(* Logix 5000 project; controller PBS_Perfusion vendor 1 type 14 code 217 rev 32.14; software revision 32.03; part 23 of 27 *)
(* tags used below, declared in another part *)
   Ref_FaultCodeList : P_DescList[1];   // Tag containing List of Fault Codes (DINT) and their Descriptions (STRING)
   Inp_LastFaultCode : DINT;   // Most recent drive fault code (enumeration)
   Inp_Ready : BOOL;   // 1=Drive is ready to run
   Inp_CommandDir : BOOL;   // 1=Drive is commanded Forward, 0=Drive is commanded Reverse
   Inp_IOFault : BOOL;   // Input Communication Status 0=OK, 1=fail
   Inp_Sim : BOOL;   // 1=Simulate working drive; 0=Start/Stop/ Monitor actual drive
   Cfg_HasReverse : BOOL;   // 1=Drive can be run reverse, 0=Forward only
   Cfg_HasJog : BOOL;   // 1=Drive Jog Command enabled/visible, 0=Drive Jog Command not allowed
   Cfg_HasRunFdbk : BOOL;   // 1=Drive provides feedback signal on Inp_Running when running
   Cfg_HasSpeedFdbk : BOOL;   // 1=Drive provides speed feedback on Inp_SpeedFdbk
   Cfg_UseSpeedFdbk : BOOL;   // 1=Drive speed determines running state, 0=state determined by drive Active input bit
   Cfg_HasOutDatalink : BOOL;   // 1=A signal is connected to Out_Datalink
   Cfg_SetTrack : BOOL;   // 1=Settings track for unselected sources, 0=no tracking
   Cfg_SetTrackOvrdHand : BOOL;   // 1=Prog/Oper/Ext Settings track Override/Hand
   Cfg_OperStopPrio : BOOL;   // 1=OCmd_Stop any time, 0=OCmd_Stop only when Oper selected
   Cfg_OCmdResets : BOOL;   // 1=New drive OCmd resets shed latches and cleared alarms, 0=OCmdReset req'd.
   Cfg_ShedOnFailToStart : BOOL;   // 1=Stop Motor and Alarm on Fail to Start; 0=Alarm only on Fail to Start
   Cfg_MinSpdRef : REAL;   // Minimum Speed Reference in EU (for limiting)
   Cfg_MaxSpdRef : REAL;   // Maximum Speed Reference in EU (for limiting)
   Cfg_SpeedRefRawMin : REAL;   // Speed Reference Minimum in Drive (raw) Units (for scaling)
   Cfg_SpeedRefRawMax : REAL;   // Speed Reference Maximum in Drive (raw) Units (for scaling)
   Cfg_SpeedRefEUMin : REAL;   // Speed Reference Minimum in Engineering Units (for scaling)
   Cfg_SpeedRefEUMax : REAL;   // Speed Reference Maximum in Engineering Units (for scaling)
   Cfg_OutDatalinkRawMin : REAL;   // Output Datalink Minimum in Drive (raw) Units (for scaling)
   Cfg_OutDatalinkRawMax : REAL;   // Output Datalink Maximum in Drive (raw) Units (for scaling)
   Cfg_OutDatalinkEUMin : REAL;   // Output Datalink Minimum in Engineering Units (for scaling)
   Cfg_OutDatalinkEUMax : REAL;   // Output Datalink Maximum in Engineering Units (for scaling)
   Cfg_OperKeep : SINT;   // Oper keeps control in Prog / Ext: .0=Reference, .1=Start/Stop/Fwd/ Rev, .3=OutDatalink
   Cfg_ProgKeep : SINT;   // Prog keeps control in Oper / Ext: .0=Reference, .1=Start/Stop/Fwd/ Rev, .3=OutDatalink
   PSet_SpeedRef : REAL;   // Program Setting of Speed Reference (EU)
   PSet_OutDatalink : REAL;   // Program Setting of Output Datalink (EU)
   XSet_SpeedRef : REAL;   // External Setting of Speed Reference (EU)
   XSet_OutDatalink : REAL;   // External Setting of Output Datalink (EU)
   Out_SpeedRef : REAL;   // Drive Speed Reference in Drive Units (typ. 0-32767 = 0 to max freq.)
   Out_Datalink : REAL;   // Auxiliary Signal (datalink) Output in Drive (raw) Units
   Out_Run : BOOL;   // 1=Start/Run Drive, 0=Stop Drive (for held starter type)
   Out_Stop : BOOL;   // 1=Stop Drive, 0=drive left in current state
   Out_Start : BOOL;   // 1=Start Drive, 0=drive left in current state
   Out_Jog : BOOL;   // 1=Jog drive at Jog Speed, -->0=stop jogging
   Out_Fwd : BOOL;   // 1=Set drive direction to Forward
   Out_Rev : BOOL;   // 1=Set drive direction to Reverse
   Out_Horn : BOOL;   // 1=Sound audible prior to commanded motor start
   Val_SpeedRef : REAL;   // Speed Reference (target) to drive
   Val_OutDatalink : REAL;   // Output Datalink value to drive
   Val_LastFaultCode : DINT;   // Most recent drive fault code (enumeration)
   SrcQ_IO : DINT;   // Source and Quality of primary I/O (enumeration)
   SrcQ : DINT;   // Source and Quality of primary Val/Sts (enumeration)
   Val_Cmd : DINT;   // Device Command 0=None, 1=Stop, 2=StartFwd 3=StartRev 4=JogFwd 5=JogRev
   Val_Sts : DINT;   // Device Sts: 0=? 1=Stopped 2=RunFwd 3=RunRev 4=RunSlow 5=StartFwd 6=StartRev 7=StartSlow 8=JogFwd 9=JogRev 10=Stopping
   Val_Fault : DINT;   // Device Fault Status 0=None, 16=Fail to Start, 17 = Fail to Stop, 18=Drive Fault, 32=I/O Fault, 34=Config Error
   Val_NotifyAll : DINT;   // Highest Alarm prio and ack status this object + channel (enum)
   Val_UnackAlmC : DINT;   // Count of Unacknowledged Alarms
   Sts_Stopped : BOOL;   // 1=Drive requested to stop and is confirmed stopped
   Sts_StartingFwd : BOOL;   // 1=Drive requested to run forward and awaiting run feedback
   Sts_StartingRev : BOOL;   // 1=Drive requested to run reverse and awaiting run feedback
   Sts_RunningFwd : BOOL;   // 1=Drive requested to run and is confirmed running forward
   Sts_RunningRev : BOOL;   // 1=Drive requested to run and is confirmed running reverse
   Sts_StoppingFwd : BOOL;   // 1=Drive running forward requested to stop and awaiting stopped feedback
   Sts_StoppingRev : BOOL;   // 1=Drive running reverse requested to stop and awaiting stopped feedback
   Sts_JoggingFwd : BOOL;   // 1=Drive requested to Jog Forward
   Sts_JoggingRev : BOOL;   // 1=Drive requested to Jog Reverse
   Sts_Horn : BOOL;   // 1=Motor Horn Active
   Sts_CommandDir : BOOL;   // 1=Drive commanded to Forward, 0=Reverse
   Sts_ActualDir : BOOL;   // 1=Drive Actual direction is Forward, 0=Reverse
   Sts_SpeedLimited : BOOL;   // 1=Speed Reference Setting exceeds configured Max/Min limit
   Sts_NotRdy : BOOL;   // 1=Device Not Ready, see detail bits for reason
   Nrdy_CfgErr : BOOL;   // 1=Device Not Ready: Configuration Error
   Nrdy_Fail : BOOL;   // 1=Device Not Ready: Device Failure (Shed Requires Reset)
   Nrdy_IOFault : BOOL;   // 1=Device Not Ready: I/O Fault (Shed Requires Reset)
   Nrdy_PrioStop : BOOL;   // 1=Device Not Ready: Oper/Ext Priority Stop Requires Reset
   Nrdy_Trip : BOOL;   // 1=Device not Ready: Deivce Tripped (Drive Fault)
   Sts_AlmInh : BOOL;   // 1=An Alarm is Shelved, Disabled or Suppressed, display icon
   Sts_Err : BOOL;   // 1=Error in Config: see detail bits for reason
   Err_Alarm : BOOL;   // 1=Error in Config: Alarm Min On Time, Shelf Time, Severity
   Err_FdbkRaw : BOOL;   // 1=Erron in Config: Speed Fdbk Raw Min = Max
   Err_FdbkEU : BOOL;   // 1=Error in Config: Speed Fdbk EU Min = Max
   Err_RefEU : BOOL;   // 1=Error in Config: Speed Ref EU Min = Max
   Err_OutDLEU : BOOL;   // 1=Error in Config: Output Datalink EU Min = Max
   Sts_Hand : ALIAS FOR CmdSrc.Sts_Hand;
   Sts_OoS : ALIAS FOR CmdSrc.Sts_OoS;
   Sts_Maint : ALIAS FOR CmdSrc.Sts_Maint;
   Sts_Ovrd : ALIAS FOR CmdSrc.Sts_Ovrd;
   Sts_RdyReset : ALIAS FOR ORdy_Reset;   // 1=A latched alarm or shed condition is ready to be reset
   Sts_RdyAck : BOOL;   // 1=An alarm is ready to be acknowledged
   Sts_FailToStart : ALIAS FOR FailToStart.Inp;   // 1=Drive Failed to Start (One-Shot)
   Sts_FailToStop : ALIAS FOR FailToStop.Inp;   // 1=Drive Failed to Stop
   Sts_DriveFault : ALIAS FOR DriveFault.Inp;   // 1=Drive Fault (see drive display or manual)
   Sts_IOFault : ALIAS FOR IOFault.Inp;   // I/O Comm Fault Status (0=OK, 1=Bad)
   P_VSD : BOOL;   // Unique Parameter Name for auto - discovery
   CmdSrc : P_CmdSrc;   // Drive Mode Selection
   IOFault : P_Alarm;   // I/O Fault Alarm
   IntlkTrip : P_Alarm;   // Interlock Trip Alarm
   FailToStop : P_Alarm;   // Drive Failed to Stop Alarm
   FailToStart : P_Alarm;   // Drive Failed to Start Alarm
   Wrk_Run : BOOL;   // 1=Drive should be "running", 0=should be "stopped"
   Wrk_StartRetrigT : TIMER;   // Time to pulse start output on start command retrigger (Maint)
   Wrk_StopRetrigT : TIMER;   // Time to pulse stop output on stop command retrigger (Maint)
   Wrk_RunFdbk : BOOL;   // Run Feedback based on mode, simulation, etc. 1=running
   Wrk_Notify : DINT;   // Buffer for building Val_Notify
   DriveFault : P_Alarm;   // Drive Faulted Alarm
   Wrk_SpeedRef : REAL;   // Working copy of Speed Reference (for limiting)
   Wrk_Rev : BOOL;   // Working (internal) Direction 1=Reverse 0=Forward (default)
   Wrk_Jog : BOOL;   // 1=Jog Drive, 0=Drive not jogging
   Wrk_OutDatalink : REAL;   // Selected Output Datalink setting
   Wrk_StopT : TIMER;   // Stop Check Timer (for Fail to Stop)
   Wrk_StartT : TIMER;   // Start Check Timer (for Fail to Start)
   Wrk_Cmd : DINT;   // Buffer for building Val_Cmd
   Wrk_Sts : DINT;   // Buffer for building Val_Sts
   Wrk_Fault : DINT;   // Buffer for building Val_Fault
   Wrk_Retrigger : BOOL;   // Maint Start issued while running or Stop while stopped
   Wrk_JogT : TIMER;   // Jog Timer
   Wrk_FaultDescFSC : CONTROL;   // FSC control for Fault Code List search
   Val_FaultDesc : STRING_40;   // Description of Drive Fault (given LastFaultCode)
   Wrk_SrcQ : DINT;   // Register for building Source / Quality enumeration
   Val_Notify : DINT;   // Current Alarm Level and Acknowledgement (enumeration)
   Wrk_NotRdy : BOOL;   // Device Not Ready conditions excluding shed latches
   Wrk_StartInhT : TIMER;   // Local Start Inhibit Timer
   Wrk_StopInhT : TIMER;   // Local Stop Inhibit Timer
   Wrk_Hand : BOOL;   // Perform Hand Mode alignment with actual device state
   Wrk_UnackAlmC : DINT;   // Buffer for building Val_UnackAlmC
   Wrk_StartHornT : TIMER;   // Timer for audible alert or start
   Wrk_StartHorn : BOOL;   // 1=Sound audible prior to commanded motor start
   Wrk_RevPermOK : BOOL;   // Reverse Permissives and NB Permissive OK
   Wrk_FwdPermOK : BOOL;   // Forward Permissives and NB Permissive OK
   OSet_OutDatalink : REAL;   // Operator Setting of Output Datalink (EU)
   OSet_SpeedRef : REAL;   // Operator Setting of Speed Reference (EU)
   ORdy_ResetAckAll : BOOL;   // 1=Ready for OCmd_ResetAckAll (enables HMI button)
   ORdy_Reset : BOOL;   // 1=Ready for OCmd_Reset (enables HMI button)
   ORdy_JogRev : BOOL;   // 1=Ready for OCmd_JogRev (enabled HMI button)
   ORdy_JogFwd : BOOL;   // 1=Ready for OCmd_JogFwd (enables HMI button)
   ORdy_Stop : BOOL;   // 1=Ready for OCmd_Stop (enables HMI button)
   ORdy_StartRev : BOOL;   // 1=Ready for OCmd_StartRev (enables HMI button)
   ORdy_StartFwd : BOOL;   // 1=Ready for OCmd_StartFwd (enables HMI button)
   Wrk_OperHas1 : BOOL;   // Operator has Commands
   REAL : DINT;
(* P_VSD, continued *)

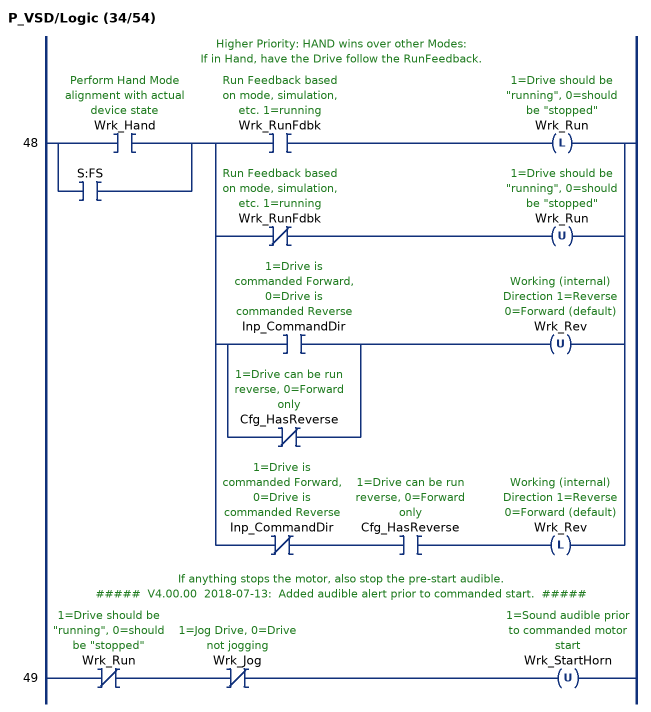
   [picture p515: P_VSD/Logic rungs 48-49]
   // Higher Priority: HAND wins over other Modes:
   // If in Hand, have the Drive follow the RunFeedback.
   48: [XIC(Wrk_Hand) ,XIC(S:FS) ][XIC(Wrk_RunFdbk) OTL(Wrk_Run) ,XIO(Wrk_RunFdbk) OTU(Wrk_Run) ,[XIC(Inp_CommandDir) ,XIO(Cfg_HasReverse) ] OTU(Wrk_Rev) ,XIO(Inp_CommandDir) XIC(Cfg_HasReverse) OTL(Wrk_Rev) ];
   // If anything stops the motor, also stop the pre-start audible.
   // #####  V4.00.00  2018-07-13:  Added audible alert prior to commanded start.  #####
   49: XIO(Wrk_Run)XIO(Wrk_Jog)OTU(Wrk_StartHorn);
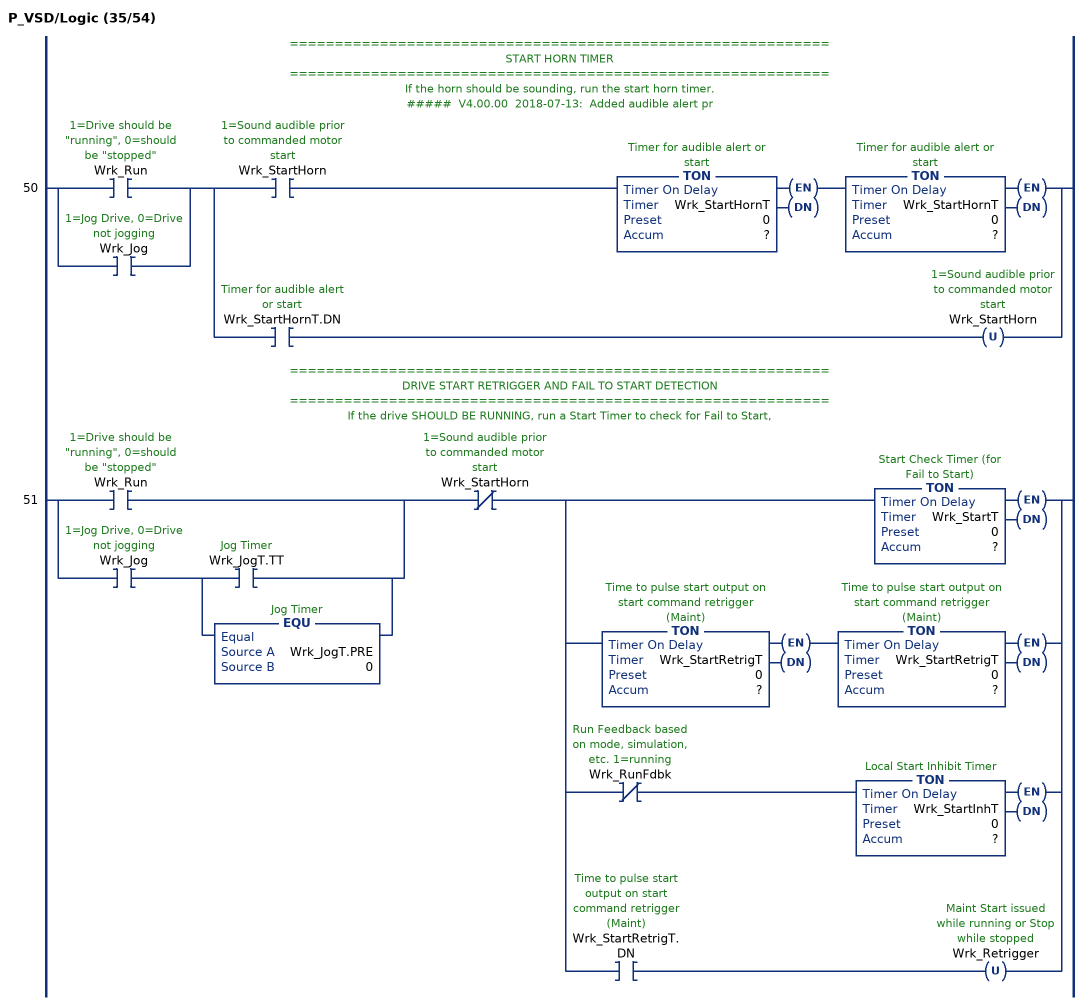
   // ============================================================
   // START HORN TIMER
   // ============================================================
   // If the horn should be sounding, run the start horn timer.
   // #####  V4.00.00  2018-07-13:  Added audible alert pr
   50: [XIC(Wrk_Run) ,XIC(Wrk_Jog) ][XIC(Wrk_StartHorn) TON(Wrk_StartHornT,?,?) TON(Wrk_StartHornT,?,?) ,XIC(Wrk_StartHornT.DN) OTU(Wrk_StartHorn) ];
   // ============================================================
   // DRIVE START RETRIGGER AND FAIL TO START DETECTION
   // ============================================================
   // If the drive SHOULD BE RUNNING, run a Start Timer to check for Fail to Start,
   51: [XIC(Wrk_Run) ,XIC(Wrk_Jog) [XIC(Wrk_JogT.TT) ,EQU(Wrk_JogT.PRE,0) ] ]XIO(Wrk_StartHorn)[TON(Wrk_StartT,?,?) ,TON(Wrk_StartRetrigT,?,?) TON(Wrk_StartRetrigT,?,?) ,XIO(Wrk_RunFdbk) TON(Wrk_StartInhT,?,?) ,XIC(Wrk_StartRetrigT.DN) OTU(Wrk_Retrigger) ];
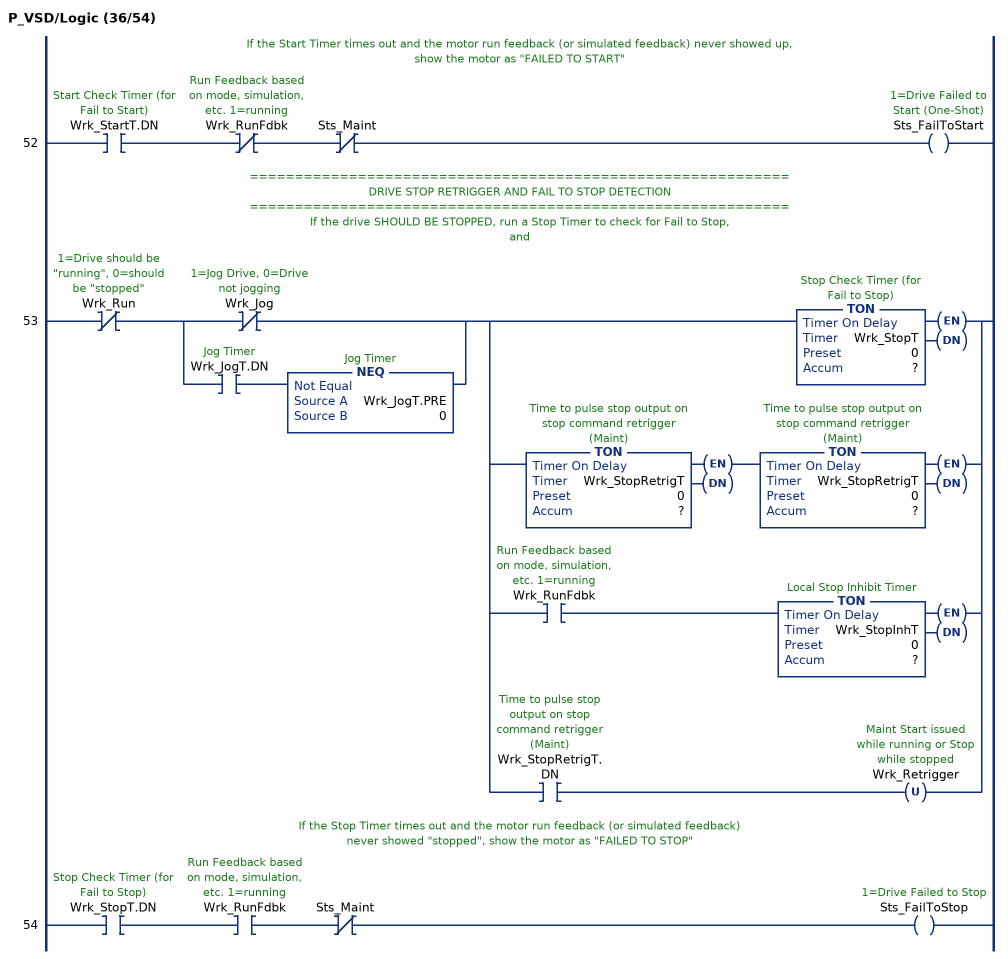
   // If the Start Timer times out and the motor run feedback (or simulated feedback) never showed up,
   // show the motor as "FAILED TO START"
   52: XIC(Wrk_StartT.DN)XIO(Wrk_RunFdbk)XIO(Sts_Maint)OTE(Sts_FailToStart);
   // ============================================================
   // DRIVE STOP RETRIGGER AND FAIL TO STOP DETECTION
   // ============================================================
   // If the drive SHOULD BE STOPPED, run a Stop Timer to check for Fail to Stop,
   //  and
   53: XIO(Wrk_Run)[XIO(Wrk_Jog) ,XIC(Wrk_JogT.DN) NEQ(Wrk_JogT.PRE,0) ][TON(Wrk_StopT,?,?) ,TON(Wrk_StopRetrigT,?,?) TON(Wrk_StopRetrigT,?,?) ,XIC(Wrk_RunFdbk) TON(Wrk_StopInhT,?,?) ,XIC(Wrk_StopRetrigT.DN) OTU(Wrk_Retrigger) ];
   // If the Stop Timer times out and the motor run feedback (or simulated feedback)
   // never showed "stopped", show the motor as "FAILED TO STOP"
   54: XIC(Wrk_StopT.DN)XIC(Wrk_RunFdbk)XIO(Sts_Maint)OTE(Sts_FailToStop);
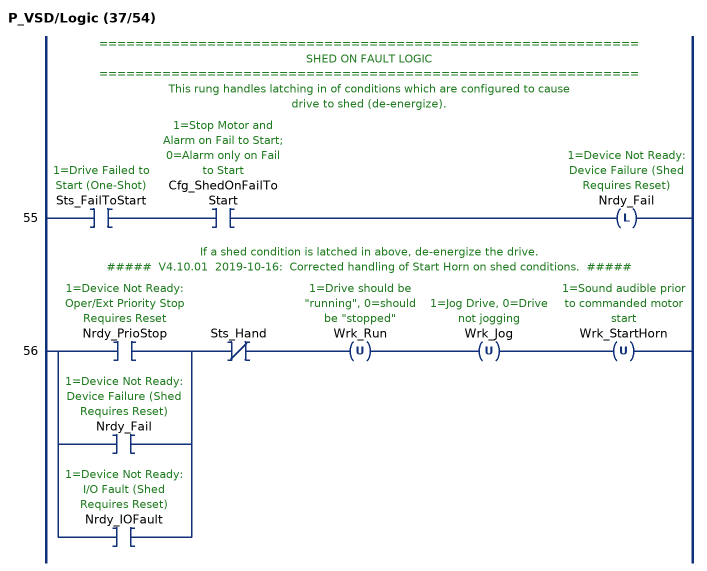
   // ============================================================
   // SHED ON FAULT LOGIC
   // ============================================================
   // This rung handles latching in of conditions which are configured to cause
   // drive to shed (de-energize).
   55: XIC(Sts_FailToStart)XIC(Cfg_ShedOnFailToStart)OTL(Nrdy_Fail);
   // If a shed condition is latched in above, de-energize the drive.
   // #####  V4.10.01  2019-10-16:  Corrected handling of Start Horn on shed conditions.  #####
   56: [XIC(Nrdy_PrioStop) ,XIC(Nrdy_Fail) ,XIC(Nrdy_IOFault) ]XIO(Sts_Hand)OTU(Wrk_Run)OTU(Wrk_Jog)OTU(Wrk_StartHorn);
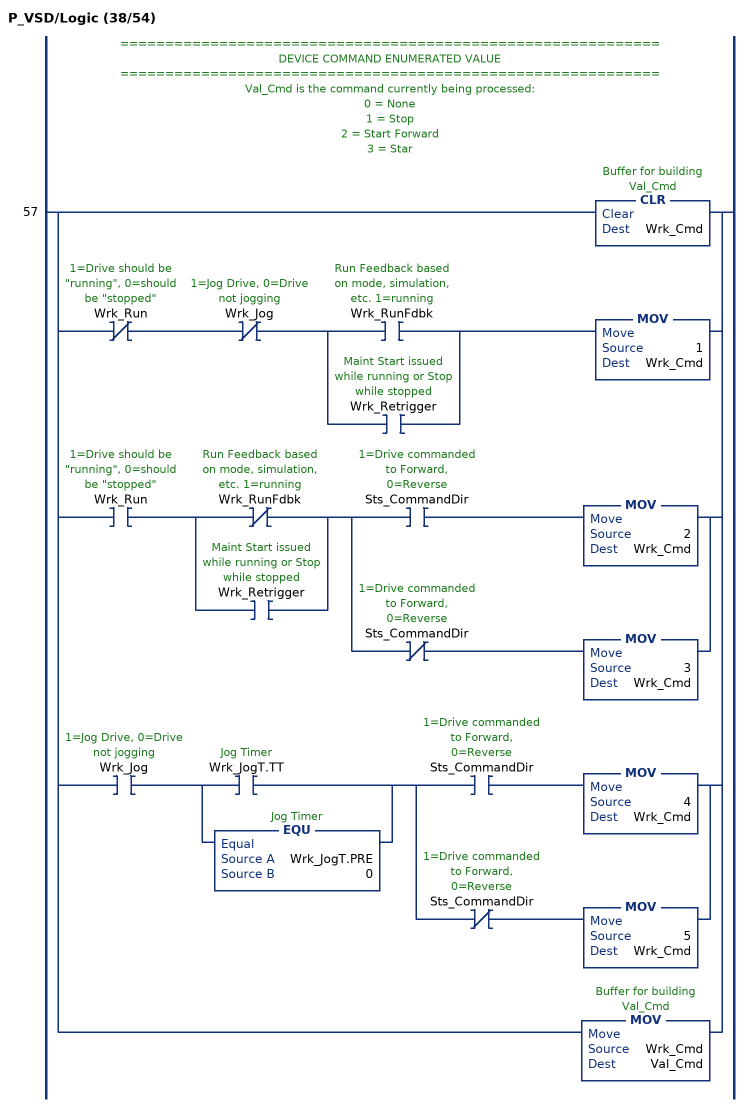
   // ============================================================
   // DEVICE COMMAND ENUMERATED VALUE
   // ============================================================
   // Val_Cmd is the command currently being processed:
   // 0 = None
   // 1 = Stop
   // 2 = Start Forward
   // 3 = Star
   57: [CLR(Wrk_Cmd) ,XIO(Wrk_Run) XIO(Wrk_Jog) [XIC(Wrk_RunFdbk) ,XIC(Wrk_Retrigger) ] MOV(1,Wrk_Cmd) ,XIC(Wrk_Run) [XIO(Wrk_RunFdbk) ,XIC(Wrk_Retrigger) ] [XIC(Sts_CommandDir) MOV(2,Wrk_Cmd) ,XIO(Sts_CommandDir) MOV(3,Wrk_Cmd) ] ,XIC(Wrk_Jog) [XIC(Wrk_JogT.TT) ,EQU(Wrk_JogT.PRE,0) ] [XIC(Sts_CommandDir) MOV(4,Wrk_Cmd) ,XIO(Sts_CommandDir) MOV(5,Wrk_Cmd) ] ,MOV(Wrk_Cmd,Val_Cmd) ];
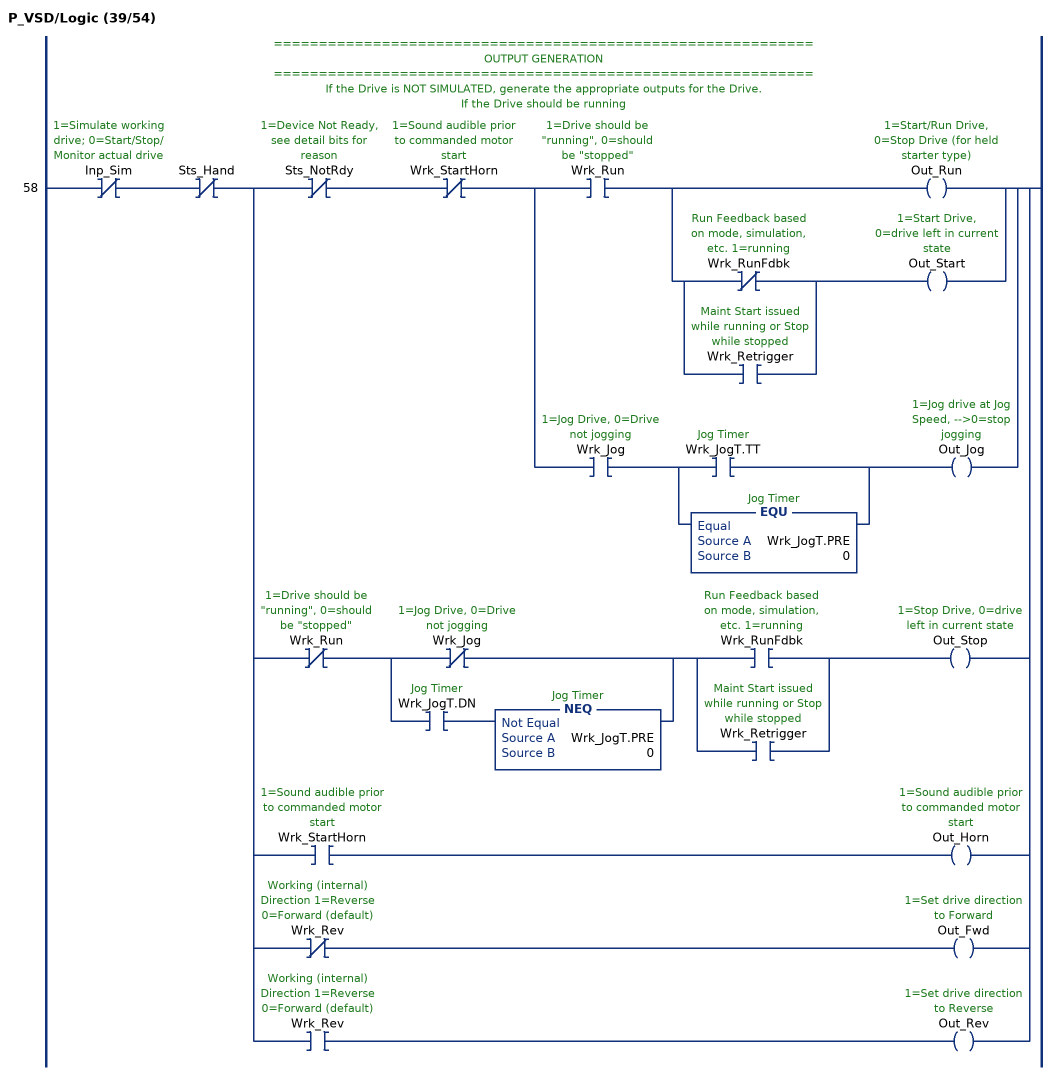
   // ============================================================
   // OUTPUT GENERATION
   // ============================================================
   // If the Drive is NOT SIMULATED, generate the appropriate outputs for the Drive.
   // If the Drive should be running
   58: XIO(Inp_Sim)XIO(Sts_Hand)[XIO(Sts_NotRdy) XIO(Wrk_StartHorn) [XIC(Wrk_Run) [OTE(Out_Run) ,[XIO(Wrk_RunFdbk) ,XIC(Wrk_Retrigger) ] OTE(Out_Start) ] ,XIC(Wrk_Jog) [XIC(Wrk_JogT.TT) ,EQU(Wrk_JogT.PRE,0) ] OTE(Out_Jog) ] ,XIO(Wrk_Run) [XIO(Wrk_Jog) ,XIC(Wrk_JogT.DN) NEQ(Wrk_JogT.PRE,0) ] [XIC(Wrk_RunFdbk) ,XIC(Wrk_Retrigger) ] OTE(Out_Stop) ,XIC(Wrk_StartHorn) OTE(Out_Horn) ,XIO(Wrk_Rev) OTE(Out_Fwd) ,XIC(Wrk_Rev) OTE(Out_Rev) ];
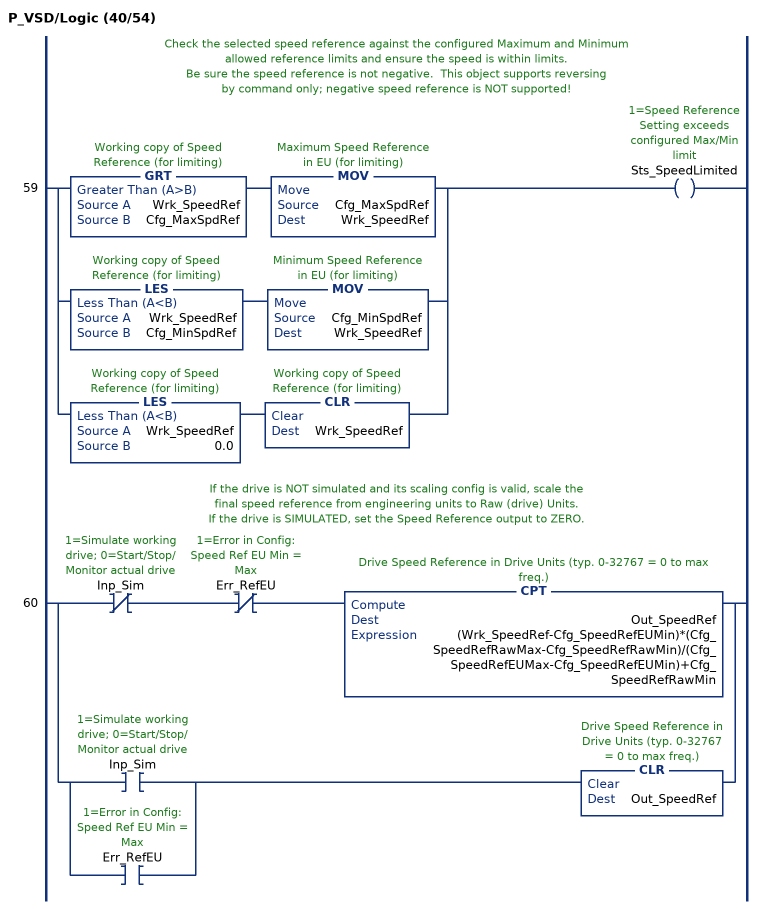
   // Check the selected speed reference against the configured Maximum and Minimum
   // allowed reference limits and ensure the speed is within limits.
   // Be sure the speed reference is not negative.  This object supports reversing
   // by command only; negative speed reference is NOT supported!
   59: [GRT(Wrk_SpeedRef,Cfg_MaxSpdRef) MOV(Cfg_MaxSpdRef,Wrk_SpeedRef) ,LES(Wrk_SpeedRef,Cfg_MinSpdRef) MOV(Cfg_MinSpdRef,Wrk_SpeedRef) ,LES(Wrk_SpeedRef,0.0) CLR(Wrk_SpeedRef) ]OTE(Sts_SpeedLimited);
   // If the drive is NOT simulated and its scaling config is valid, scale the
   // final speed reference from engineering units to Raw (drive) Units.
   // If the drive is SIMULATED, set the Speed Reference output to ZERO.
   60: [XIO(Inp_Sim) XIO(Err_RefEU) CPT(Out_SpeedRef,(Wrk_SpeedRef-Cfg_SpeedRefEUMin)*(Cfg_SpeedRefRawMax-Cfg_SpeedRefRawMin)/(Cfg_SpeedRefEUMax-Cfg_SpeedRefEUMin)+Cfg_SpeedRefRawMin) ,[XIC(Inp_Sim) ,XIC(Err_RefEU) ] CLR(Out_SpeedRef) ];
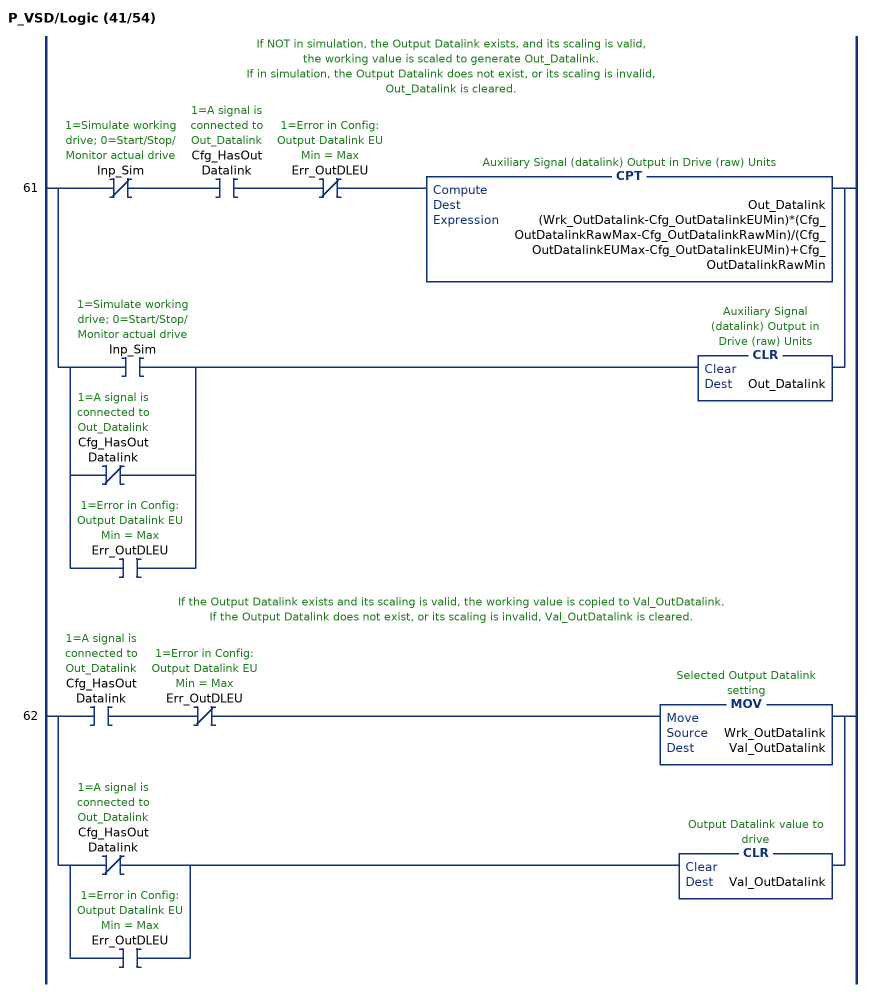
   // If NOT in simulation, the Output Datalink exists, and its scaling is valid,
   // the working value is scaled to generate Out_Datalink.
   // If in simulation, the Output Datalink does not exist, or its scaling is invalid,
   // Out_Datalink is cleared.
   61: [XIO(Inp_Sim) XIC(Cfg_HasOutDatalink) XIO(Err_OutDLEU) CPT(Out_Datalink,(Wrk_OutDatalink-Cfg_OutDatalinkEUMin)*(Cfg_OutDatalinkRawMax-Cfg_OutDatalinkRawMin)/(Cfg_OutDatalinkEUMax-Cfg_OutDatalinkEUMin)+Cfg_OutDatalinkRawMin) ,[XIC(Inp_Sim) ,XIO(Cfg_HasOutDatalink) ,XIC(Err_OutDLEU) ] CLR(Out_Datalink) ];
   // If the Output Datalink exists and its scaling is valid, the working value is copied to Val_OutDatalink.
   // If the Output Datalink does not exist, or its scaling is invalid, Val_OutDatalink is cleared.
   62: [XIC(Cfg_HasOutDatalink) XIO(Err_OutDLEU) MOV(Wrk_OutDatalink,Val_OutDatalink) ,[XIO(Cfg_HasOutDatalink) ,XIC(Err_OutDLEU) ] CLR(Val_OutDatalink) ];
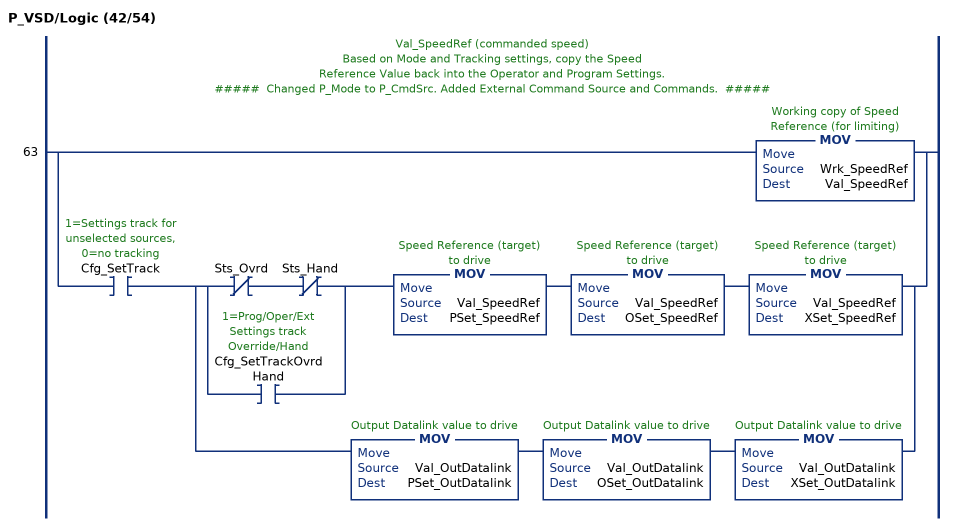
   // Val_SpeedRef (commanded speed)
   // Based on Mode and Tracking settings, copy the Speed
   // Reference Value back into the Operator and Program Settings.
   // #####  Changed P_Mode to P_CmdSrc. Added External Command Source and Commands.  #####
   63: [MOV(Wrk_SpeedRef,Val_SpeedRef) ,XIC(Cfg_SetTrack) [[XIO(Sts_Ovrd) XIO(Sts_Hand) ,XIC(Cfg_SetTrackOvrdHand) ] MOV(Val_SpeedRef,PSet_SpeedRef) MOV(Val_SpeedRef,OSet_SpeedRef) MOV(Val_SpeedRef,XSet_SpeedRef) ,MOV(Val_OutDatalink,PSet_OutDatalink) MOV(Val_OutDatalink,OSet_OutDatalink) MOV(Val_OutDatalink,XSet_OutDatalink) ] ];
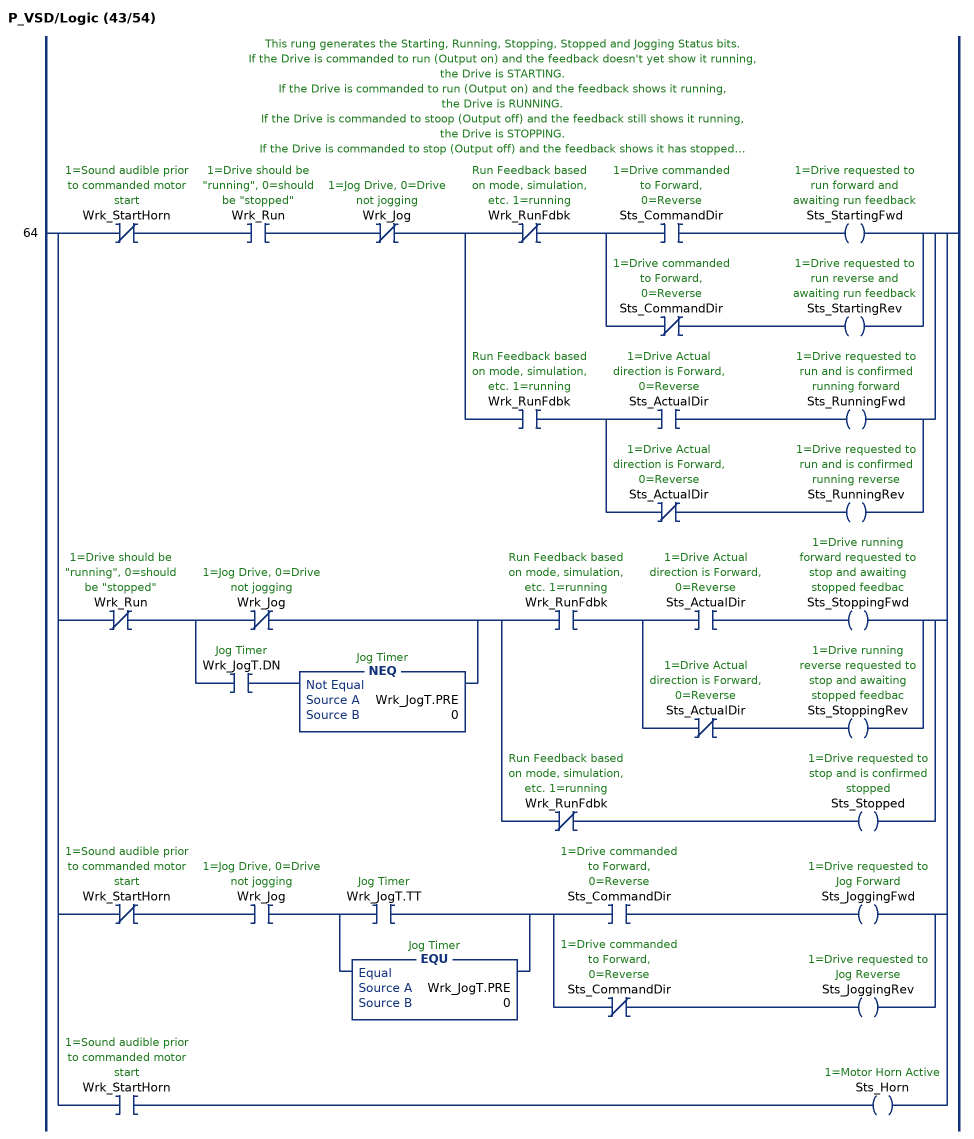
   // This rung generates the Starting, Running, Stopping, Stopped and Jogging Status bits.
   // If the Drive is commanded to run (Output on) and the feedback doesn't yet show it running,
   // the Drive is STARTING.
   // If the Drive is commanded to run (Output on) and the feedback shows it running,
   // the Drive is RUNNING.
   // If the Drive is commanded to stoop (Output off) and the feedback still shows it running,
   // the Drive is STOPPING.
   // If the Drive is commanded to stop (Output off) and the feedback shows it has stopped,
   // the Drive is STOPPED.
   // If the Drive is commanded to jog, show the status as JOGGING.
   // If the audible alert is active, show the Status as HORN.
   // #####  V4.00.00 2018-07-13:  Changed Start / Stop / Jog / Fwd / Rev to StartFwd / StartRev / Stop / JogFwd / JogRev  #####
   // #####  V4.10.00  2019-03-25:  Added Horn Status.  #####
   // #####  V4.10.01  2019-10-16:  Modified to lock out jog when jog time expires until jog commands are cleared.  #####
   64: [XIO(Wrk_StartHorn) XIC(Wrk_Run) XIO(Wrk_Jog) [XIO(Wrk_RunFdbk) [XIC(Sts_CommandDir) OTE(Sts_StartingFwd) ,XIO(Sts_CommandDir) OTE(Sts_StartingRev) ] ,XIC(Wrk_RunFdbk) [XIC(Sts_ActualDir) OTE(Sts_RunningFwd) ,XIO(Sts_ActualDir) OTE(Sts_RunningRev) ] ] ,XIO(Wrk_Run) [XIO(Wrk_Jog) ,XIC(Wrk_JogT.DN) NEQ(Wrk_JogT.PRE,0) ] [XIC(Wrk_RunFdbk) [XIC(Sts_ActualDir) OTE(Sts_StoppingFwd) ,XIO(Sts_ActualDir) OTE(Sts_StoppingRev) ] ,XIO(Wrk_RunFdbk) OTE(Sts_Stopped) ] ,XIO(Wrk_StartHorn) XIC(Wrk_Jog) [XIC(Wrk_JogT.TT) ,EQU(Wrk_JogT.PRE,0) ] [XIC(Sts_CommandDir) OTE(Sts_JoggingFwd) ,XIO(Sts_CommandDir) OTE(Sts_JoggingRev) ] ,XIC(Wrk_StartHorn) OTE(Sts_Horn) ];
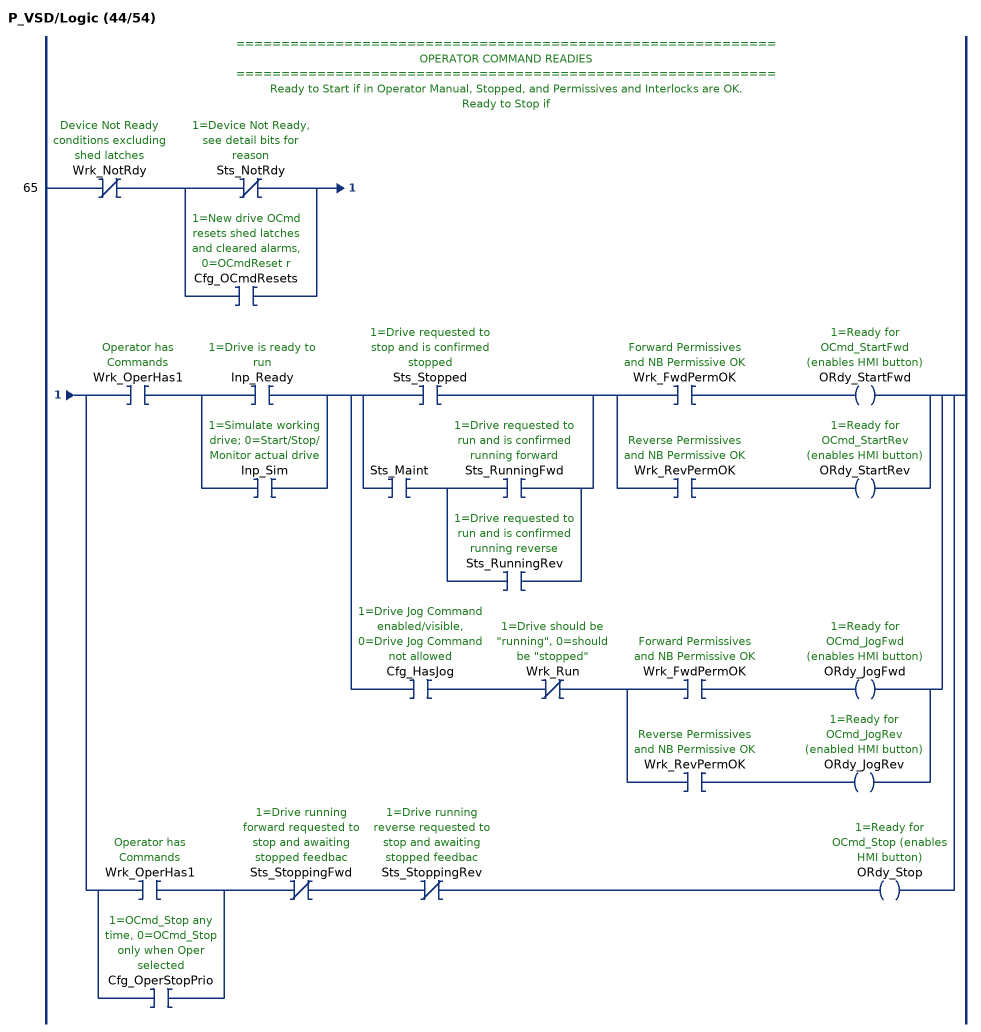
   // ============================================================
   // OPERATOR COMMAND READIES
   // ============================================================
   // Ready to Start if in Operator Manual, Stopped, and Permissives and Interlocks are OK.
   // Ready to Stop if
   65: XIO(Wrk_NotRdy)[XIO(Sts_NotRdy) ,XIC(Cfg_OCmdResets) ][XIC(Wrk_OperHas1) [XIC(Inp_Ready) ,XIC(Inp_Sim) ] [[XIC(Sts_Stopped) ,XIC(Sts_Maint) [XIC(Sts_RunningFwd) ,XIC(Sts_RunningRev) ] ] [XIC(Wrk_FwdPermOK) OTE(ORdy_StartFwd) ,XIC(Wrk_RevPermOK) OTE(ORdy_StartRev) ] ,XIC(Cfg_HasJog) XIO(Wrk_Run) [XIC(Wrk_FwdPermOK) OTE(ORdy_JogFwd) ,XIC(Wrk_RevPermOK) OTE(ORdy_JogRev) ] ] ,[XIC(Wrk_OperHas1) ,XIC(Cfg_OperStopPrio) ] XIO(Sts_StoppingFwd) XIO(Sts_StoppingRev) OTE(ORdy_Stop) ];
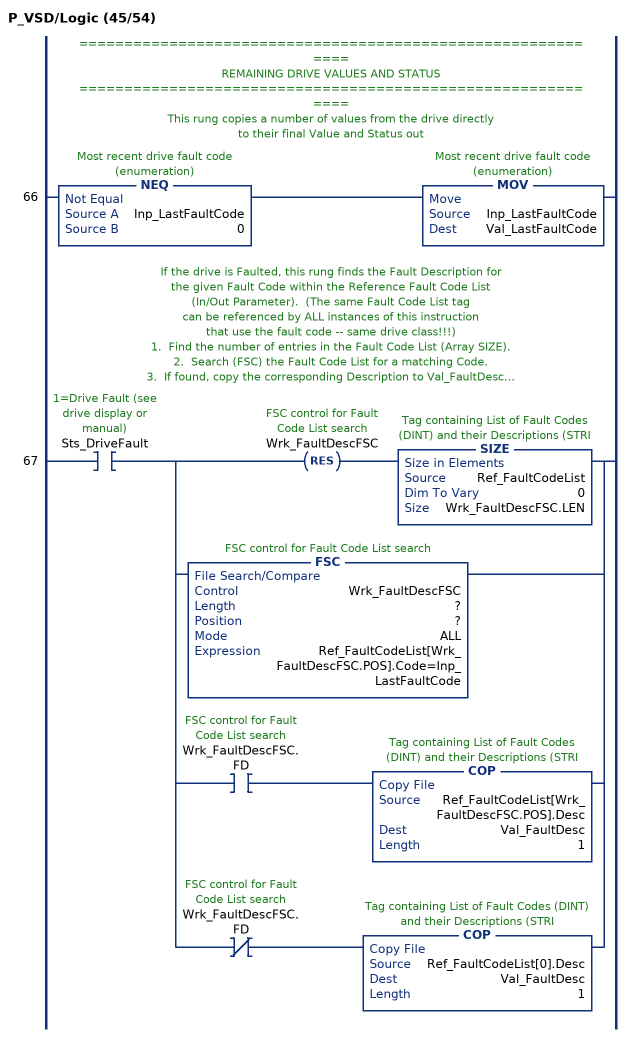
   // ============================================================
   // REMAINING DRIVE VALUES AND STATUS
   // ============================================================
   // This rung copies a number of values from the drive directly
   // to their final Value and Status out
   66: NEQ(Inp_LastFaultCode,0)MOV(Inp_LastFaultCode,Val_LastFaultCode);
   // If the drive is Faulted, this rung finds the Fault Description for
   // the given Fault Code within the Reference Fault Code List
   // (In/Out Parameter).  (The same Fault Code List tag
   // can be referenced by ALL instances of this instruction
   // that use the fault code -- same drive class!!!)
   // 1.  Find the number of entries in the Fault Code List (Array SIZE).
   // 2.  Search (FSC) the Fault Code List for a matching Code.
   // 3.  If found, copy the corresponding Description to Val_FaultDesc.
   // 4.  If NOT found, copy list entry zero ("No Help Available for this code").
   67: XIC(Sts_DriveFault)[RES(Wrk_FaultDescFSC) SIZE(Ref_FaultCodeList,0,Wrk_FaultDescFSC.LEN) ,FSC(Wrk_FaultDescFSC,?,?,ALL,Ref_FaultCodeList[Wrk_FaultDescFSC.POS].Code=Inp_LastFaultCode) ,XIC(Wrk_FaultDescFSC.FD) COP(Ref_FaultCodeList[Wrk_FaultDescFSC.POS].Desc,Val_FaultDesc,1) ,XIO(Wrk_FaultDescFSC.FD) COP(Ref_FaultCodeList[0].Desc,Val_FaultDesc,1) ];
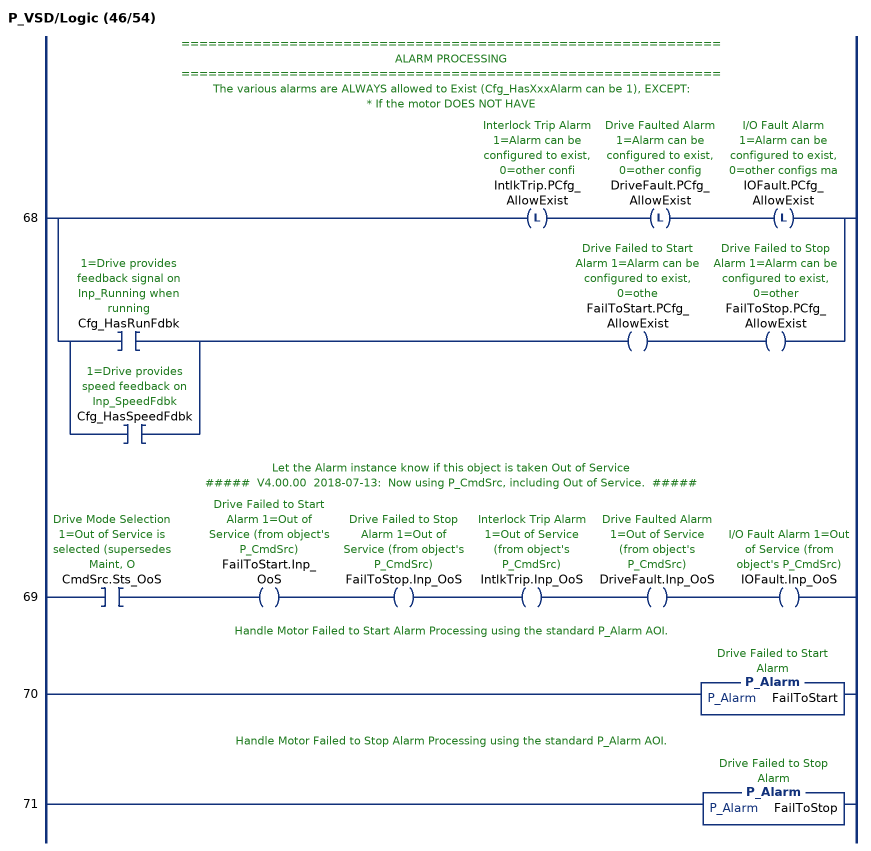
   // ============================================================
   // ALARM PROCESSING
   // ============================================================
   // The various alarms are ALWAYS allowed to Exist (Cfg_HasXxxAlarm can be 1), EXCEPT:
   // * If the motor DOES NOT HAVE
   68: [OTL(IntlkTrip.PCfg_AllowExist) OTL(DriveFault.PCfg_AllowExist) OTL(IOFault.PCfg_AllowExist) ,[XIC(Cfg_HasRunFdbk) ,XIC(Cfg_HasSpeedFdbk) ] OTE(FailToStart.PCfg_AllowExist) OTE(FailToStop.PCfg_AllowExist) ];
   // Let the Alarm instance know if this object is taken Out of Service
   // #####  V4.00.00  2018-07-13:  Now using P_CmdSrc, including Out of Service.  #####
   69: XIC(CmdSrc.Sts_OoS)OTE(FailToStart.Inp_OoS)OTE(FailToStop.Inp_OoS)OTE(IntlkTrip.Inp_OoS)OTE(DriveFault.Inp_OoS)OTE(IOFault.Inp_OoS);
   // Handle Motor Failed to Start Alarm Processing using the standard P_Alarm AOI.
   70: P_Alarm(FailToStart);
   // Handle Motor Failed to Stop Alarm Processing using the standard P_Alarm AOI.
   71: P_Alarm(FailToStop);
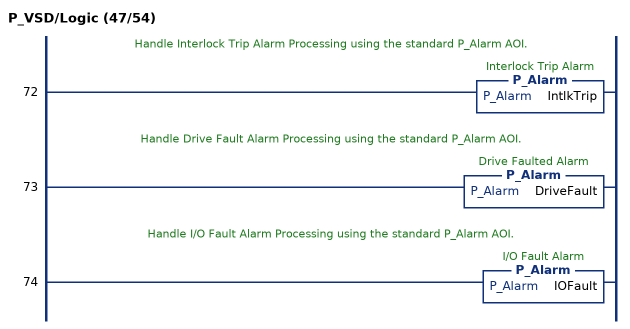
   // Handle Interlock Trip Alarm Processing using the standard P_Alarm AOI.
   72: P_Alarm(IntlkTrip);
   // Handle Drive Fault Alarm Processing using the standard P_Alarm AOI.
   73: P_Alarm(DriveFault);
   // Handle I/O Fault Alarm Processing using the standard P_Alarm AOI.
   74: P_Alarm(IOFault);
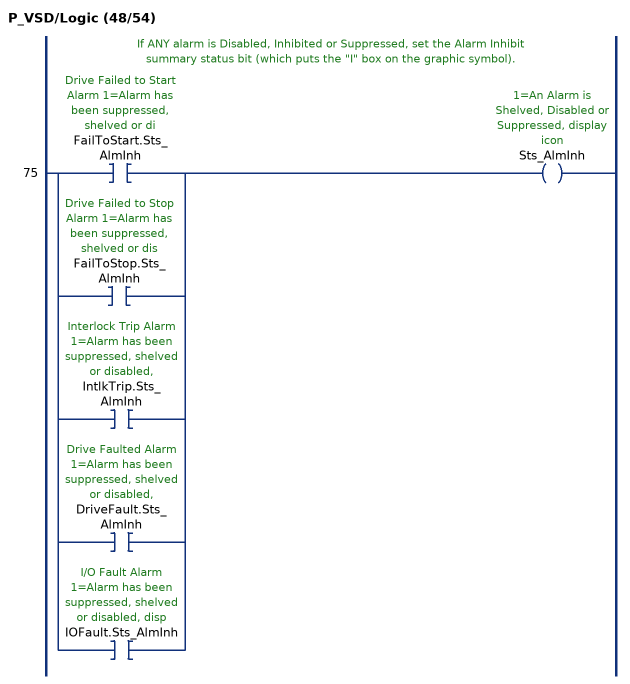
   // If ANY alarm is Disabled, Inhibited or Suppressed, set the Alarm Inhibit
   // summary status bit (which puts the "I" box on the graphic symbol).
   75: [XIC(FailToStart.Sts_AlmInh) ,XIC(FailToStop.Sts_AlmInh) ,XIC(IntlkTrip.Sts_AlmInh) ,XIC(DriveFault.Sts_AlmInh) ,XIC(IOFault.Sts_AlmInh) ]OTE(Sts_AlmInh);
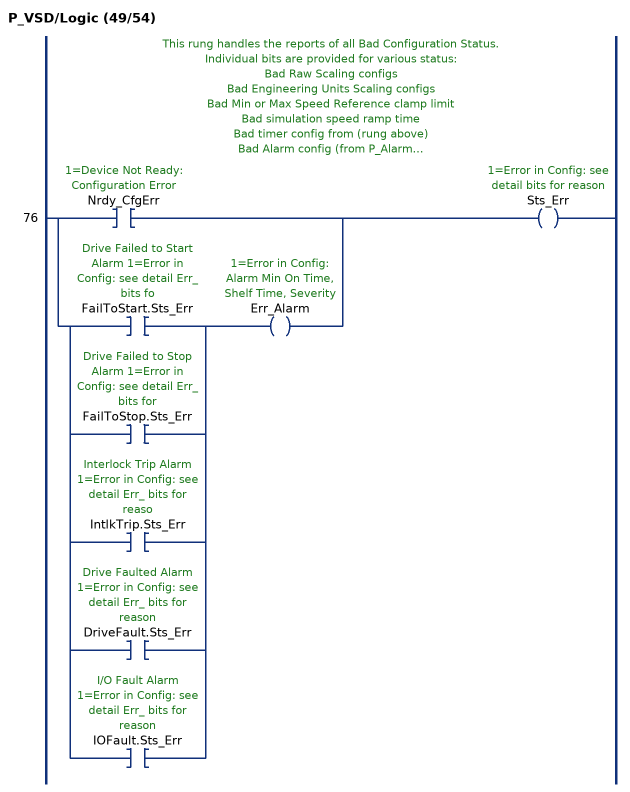
   // This rung handles the reports of all Bad Configuration Status.
   // Individual bits are provided for various status:
   // Bad Raw Scaling configs
   // Bad Engineering Units Scaling configs
   // Bad Min or Max Speed Reference clamp limit
   // Bad simulation speed ramp time
   // Bad timer config from (rung above)
   // Bad Alarm config (from P_Alarm)
   // Bad Cfg_OperKeep / Cfg_ProgKeep config
   // Then a summary Bad Config status is provided, simply an OR of the individual bits.
   // #####  V4.00.00  2018-07-13:  Modified to allow the special case where min and max clamping  #####
   // #####  limits (speed or output datalink) can be EQUAL (clamp at a specific value).  #####
   // #####  Changed delay / time configuration items to REAL seconds.  #####
   76: [XIC(Nrdy_CfgErr) ,[XIC(FailToStart.Sts_Err) ,XIC(FailToStop.Sts_Err) ,XIC(IntlkTrip.Sts_Err) ,XIC(DriveFault.Sts_Err) ,XIC(IOFault.Sts_Err) ] OTE(Err_Alarm) ]OTE(Sts_Err);
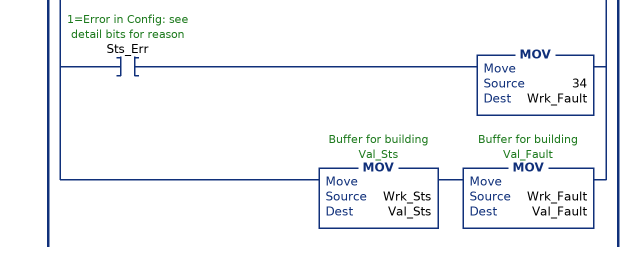
   // Val_Sts is the current device status, as determined by this AOI,
   // based on its knowledge of commands executed and feedback.
   // (This is the status that should be monitored by, for example, FT Historian.)
   // 0 = Powerup / Unknown (in Hand but having no feedback, for example)
   // 0 = Powerup / Unknown
   // 1 = Stopped
   // 2 = Running Forward
   // 3 = Running Reverse
   // 4 = Running Slow
   // 5 = Starting Forward
   // 6 = Starting Reverse
   // 7 = Starting Slow
   // 8 = Jogging Forward
   // 9 = Jogging Reverse
   // 10 = Stopping
   // 14 = Horn
   // Val_Fault is the current device fault status, as determined by this AOI,
   // based on its knowledge of commands executed and feedback.
   // (This is the fault status that should be monitored by, for example, FT Historian.)
   // 0 = None
   // 16 = Fail to Start
   // 17 = Fail to Stop
   // 18 = Drive Fault
   // 32 = I/O Fault (from Input)
   // 34 = Configuration Error
   // #####  V4.00.00 2018-07-13:  Changed Start / Stop / Jog / Fwd / Rev to StartFwd / StartRev / Stop / JogFwd / JogRev  #####
   // #####  Disable/Enable replaced by P_CmdSrc Out of Service (OoS).  #####
   // #####  V4.10.00  2019-03-25:  Added Horn Status.  #####
   77: [CLR(Wrk_Sts) CLR(Wrk_Fault) ,XIC(Sts_Stopped) MOV(1,Wrk_Sts) ,XIC(Sts_RunningFwd) MOV(2,Wrk_Sts) ,XIC(Sts_RunningRev) MOV(3,Wrk_Sts) ,XIC(Sts_StartingFwd) MOV(5,Wrk_Sts) ,XIC(Sts_StartingRev) MOV(6,Wrk_Sts) ,XIC(Sts_JoggingFwd) MOV(8,Wrk_Sts) ,XIC(Sts_JoggingRev) MOV(9,Wrk_Sts) ,[XIC(Sts_StoppingFwd) ,XIC(Sts_StoppingRev) ] MOV(10,Wrk_Sts) ,XIC(Sts_Horn) MOV(14,Wrk_Sts) ,XIC(Nrdy_Fail) MOV(16,Wrk_Fault) ,XIC(Sts_FailToStop) MOV(17,Wrk_Fault) ,XIC(Sts_DriveFault) MOV(18,Wrk_Fault) ,[XIC(Sts_IOFault) ,XIC(Nrdy_IOFault) ] MOV(32,Wrk_Fault) ,XIC(Sts_Err) MOV(34,Wrk_Fault) ,MOV(Wrk_Sts,Val_Sts) MOV(Wrk_Fault,Val_Fault) ];
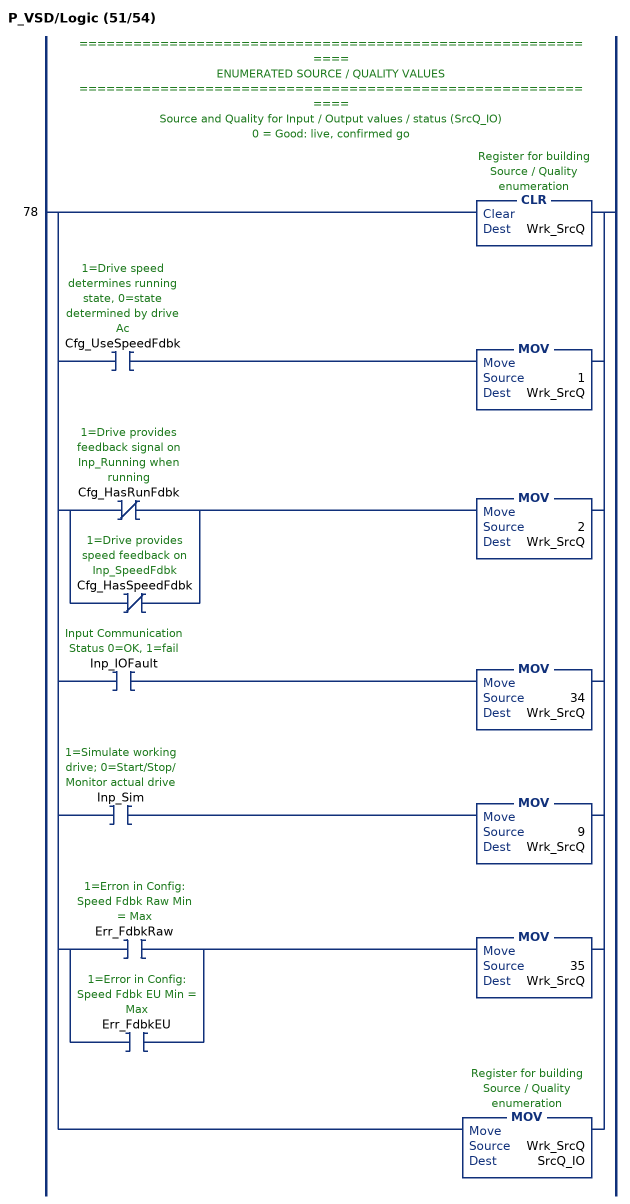
   // ============================================================
   // ENUMERATED SOURCE / QUALITY VALUES
   // ============================================================
   // Source and Quality for Input / Output values / status (SrcQ_IO)
   // 0 = Good: live, confirmed go
   78: [CLR(Wrk_SrcQ) ,XIC(Cfg_UseSpeedFdbk) MOV(1,Wrk_SrcQ) ,[XIO(Cfg_HasRunFdbk) ,XIO(Cfg_HasSpeedFdbk) ] MOV(2,Wrk_SrcQ) ,XIC(Inp_IOFault) MOV(34,Wrk_SrcQ) ,XIC(Inp_Sim) MOV(9,Wrk_SrcQ) ,[XIC(Err_FdbkRaw) ,XIC(Err_FdbkEU) ] MOV(35,Wrk_SrcQ) ,MOV(Wrk_SrcQ,SrcQ_IO) ];
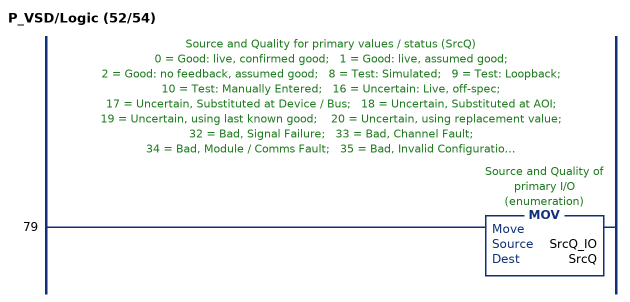
   // Source and Quality for primary values / status (SrcQ)
   // 0 = Good: live, confirmed good;   1 = Good: live, assumed good;
   // 2 = Good: no feedback, assumed good;   8 = Test: Simulated;   9 = Test: Loopback;
   // 10 = Test: Manually Entered;   16 = Uncertain: Live, off-spec;
   // 17 = Uncertain, Substituted at Device / Bus;   18 = Uncertain, Substituted at AOI;
   // 19 = Uncertain, using last known good;    20 = Uncertain, using replacement value;
   // 32 = Bad, Signal Failure;   33 = Bad, Channel Fault;
   // 34 = Bad, Module / Comms Fault;   35 = Bad, Invalid Configuration
   // If the drive is using run feedback (for state) and has speed feedback, all is live and good.
   // If the drive is using speed feedback to determine run state, state is assumed good.
   // If the drive does not have speed feedback, speed is no-feedback assumed good.
   79: MOV(SrcQ_IO,SrcQ);
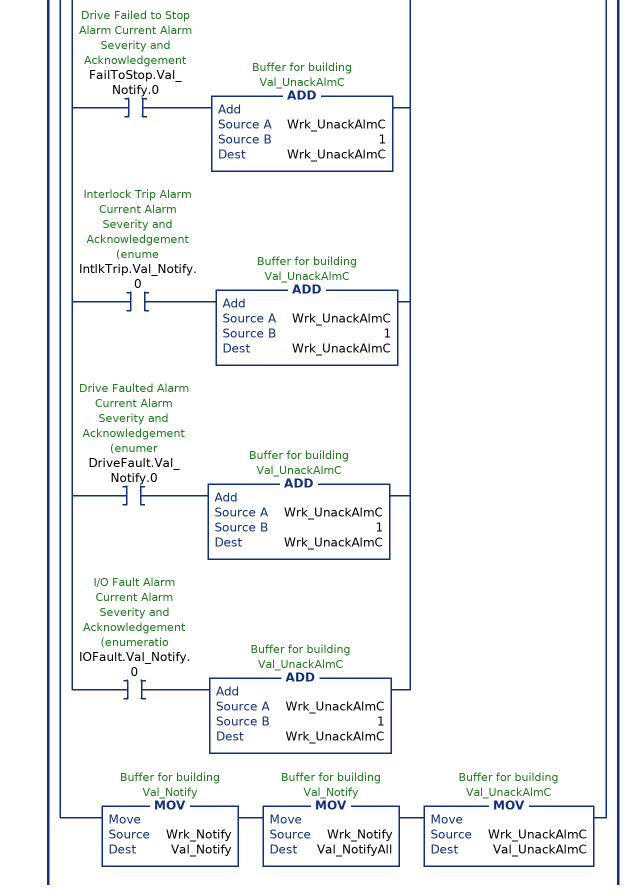
   // ============================================================
   // NOTIFICATION VALUE
   // ============================================================
   // Indicate the current alarm notification level as the max of any of the alarms,
   // and set the low-order bit for r
   80: [CLR(Wrk_Notify) CLR(Wrk_UnackAlmC) ,GRT(FailToStart.Val_Notify,Wrk_Notify) MOV(FailToStart.Val_Notify,Wrk_Notify) ,GRT(FailToStop.Val_Notify,Wrk_Notify) MOV(FailToStop.Val_Notify,Wrk_Notify) ,GRT(IntlkTrip.Val_Notify,Wrk_Notify) MOV(IntlkTrip.Val_Notify,Wrk_Notify) ,GRT(DriveFault.Val_Notify,Wrk_Notify) MOV(DriveFault.Val_Notify,Wrk_Notify) ,GRT(IOFault.Val_Notify,Wrk_Notify) MOV(IOFault.Val_Notify,Wrk_Notify) ,[XIC(FailToStart.Val_Notify.0) ADD(Wrk_UnackAlmC,1,Wrk_UnackAlmC) ,XIC(FailToStop.Val_Notify.0) ADD(Wrk_UnackAlmC,1,Wrk_UnackAlmC) ,XIC(IntlkTrip.Val_Notify.0) ADD(Wrk_UnackAlmC,1,Wrk_UnackAlmC) ,XIC(DriveFault.Val_Notify.0) ADD(Wrk_UnackAlmC,1,Wrk_UnackAlmC) ,XIC(IOFault.Val_Notify.0) ADD(Wrk_UnackAlmC,1,Wrk_UnackAlmC) ] OTE(Wrk_Notify.0) ,MOV(Wrk_Notify,Val_Notify) MOV(Wrk_Notify,Val_NotifyAll) MOV(Wrk_UnackAlmC,Val_UnackAlmC) ];
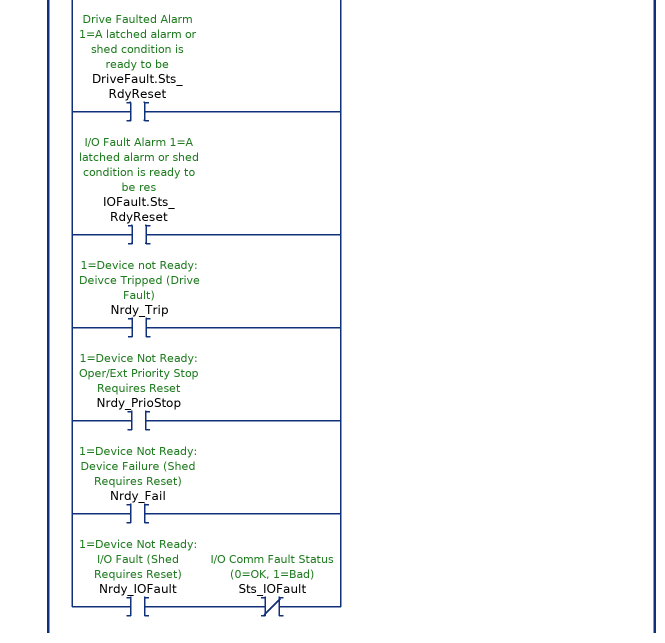
   // This rung identifies:
   // * if a latched Shed condition requires a reset in order to run the motor;
   // * if that reset or any alarm reset or other reset is required; and
   // * if any reset or acknowledge from the operator is required.
   // #####  V4.00.00  2018-07-13:  Aligned ready bit naming with command bit names.  #####
   // #####  All OCmds/MCmds and ORdys/MRdys are now Local Tags.  #####
   // #####  Added Sts_RdyAck and Sts_ResetReqd for use by external objects.  #####
   81: [[XIC(FailToStart.Sts_RdyAck) ,XIC(FailToStop.Sts_RdyAck) ,XIC(IntlkTrip.Sts_RdyAck) ,XIC(IOFault.Sts_RdyAck) ,XIC(DriveFault.Sts_RdyAck) ] OTE(Sts_RdyAck) ,[XIC(FailToStart.Sts_RdyReset) ,XIC(FailToStop.Sts_RdyReset) ,XIC(IntlkTrip.Sts_RdyReset) ,XIC(DriveFault.Sts_RdyReset) ,XIC(IOFault.Sts_RdyReset) ,XIC(Nrdy_Trip) ,XIC(Nrdy_PrioStop) ,XIC(Nrdy_Fail) ,XIC(Nrdy_IOFault) XIO(Sts_IOFault) ] OTE(ORdy_Reset) ]OTE(ORdy_ResetAckAll);
END_ROUTINE
